TYPE ST_TempLoad_Cmd :
STRUCT
	bLoadPparams: BOOL;
	bLoadMparams: BOOL;
	bLoadSupplyParams: BOOL;
END_STRUCT
END_TYPE

(* stored: Version 1.1.0.1, ProductVersion 3.1.0.26
   DUT ST_TempLoad_Cmd: Id {92d2fbfb-df73-4b23-a5f8-0cfcce48bc8f} *)
